TYPE ListLength : INT; END_TYPE

(* stored: Version 1.1.0.1, ProductVersion 3.1.4024.12
   DUT ListLength: Id {b702c7b8-eaed-4909-a174-efe76cf1dae8} *)
